// TwinCAT 3 PLC project PLC
// ProgramVersion: 3.1.4026.24
// libraries:
//   Tc2_MC2, * (Beckhoff Automation GmbH)
//   Tc2_Standard, * (Beckhoff Automation GmbH)
//   Tc2_System, * (Beckhoff Automation GmbH)
//   XPlanarApplication, * (Beckhoff Automation LLC)
// project tree:
//   / E_Steps.TcDUT, MAIN.TcPOU, PlcTask.TcTTO
//   Transformation/ ATAN2.TcPOU (not stored), MoverToWorldTransform.TcPOU
// real-time tasks:
//   TASK XPlanar Task_3: cycle T#250us, priority 1, ADS port 350
//   TASK XPlanar Task_4: cycle T#250us, priority 2, ADS port 351
//   TASK XPlanar Task_5: cycle T#250us, priority 3, ADS port 352
//   TASK Job Task: cycle default, priority 4
//   TASK MC-Task (MET): cycle T#2ms, priority 5, ADS port 353
//   TASK MC-Task (MPT): cycle T#10ms, priority 6, ADS port 354
//   TASK PlcTask: cycle T#10ms, priority 20, ADS port 355
// motion (NC):
//   TASK NC-Task 1 SAF: cycle T#2ms, priority 7, ADS port 501
//   TASK NC-Task 1 SVB: cycle T#10ms, priority 12, ADS port 511
//   AXIS CAxis (id 1)
//     Velo: SlowManual=5, FastManual=50
//     OtherSettings: AllowMotionCmdToSlave=true
//     encoder EncType=1
//     drive DrvType=5
//       Analog: TorqueSetpointScale=10, ScaleFactorActTorque=0.1
//       TimeComp: TaskDelayCycles=1
//     controller CtrType=1
//       CtrPara: PriorControlFactor=1
//         Observer: BandWidth=20
// variable links:
//   (this object) <-> NC-Task 1 SAF/Axes/CAxis
//     PlcTask Inputs/MAIN.CAxis.NcToPlc <-> Outputs/ToPlc
//     PlcTask Outputs/MAIN.CAxis.PlcToNc <-> Inputs/FromPlc
//   (this object) <-> XPlanar MC Project/Axes/Mover4330_1
//     PlcTask Inputs/MAIN.Mover._Mover.MCTOPLC/ACT <-> McToPlc/ACT
//     PlcTask Inputs/MAIN.Mover._Mover.MCTOPLC/COORDMODE <-> McToPlc/COORDMODE
//     PlcTask Inputs/MAIN.Mover._Mover.MCTOPLC/SET <-> McToPlc/SET
//     PlcTask Inputs/MAIN.Mover._Mover.MCTOPLC/SETONTRACK <-> McToPlc/SETONTRACK
//     PlcTask Inputs/MAIN.Mover._Mover.MCTOPLC/STD <-> McToPlc/STD
//     PlcTask Outputs/MAIN.Mover._Mover.PLCTOMC/STD <-> PlcToMc/STD
//   (this object) <-> XPlanar MC Project/Groups/Environment
//     PlcTask Inputs/XPlanar.Environment.MCTOPLC_STD <-> McToPlc/STD
//   (this object) <-> XPlanar MC Project/Groups/XPlanar
//     PlcTask Inputs/XPlanar.Group.MCTOPLC_STD <-> McToPlc/STD

CONFIGURATION PLC
    RESOURCE PLC ON TwinCAT3
        TASK PlcTask(INTERVAL := T#10ms, PRIORITY := 20);
        PROGRAM MAIN WITH PlcTask : MAIN;
    END_RESOURCE
END_CONFIGURATION

// ---- E_Steps.TcDUT
{attribute 'qualified_only'}
{attribute 'strict'}
{attribute 'to_string'}
TYPE E_Steps :
(
	init := 0,
    enable,
    enabled,
    moveCenter,
    idle,
    enableExtSp,
    runExtSp,
    error
)UINT;
END_TYPE

// ---- MAIN.TcPOU
PROGRAM MAIN
VAR
   MoverToWorldTransform : MoverToWorldTransform;
   XPlanarTable : FB_Component_XPlanar;
   Mover : FB_XPlanarMover;
   seq : E_Steps;
   subSeq : UDINT;
   
   Position : MoverVector;
   Velocity : MoverVector;
   Acceleration : MoverVector;
   
   CAxisPower : MC_Power;
   CAxis : AXIS_REF;
   a,b : LREAL;
   Exception : __SYSTEM.ExceptionCode;
END_VAR

CASE seq OF
    E_Steps.init:
        ip.Movers[1] := Mover;
        subSeq := 0;
        // wait for manual command to enable
        
    E_Steps.enable:
        IF XplanarTable.EnableMovers().Done THEN
            seq:= E_Steps.enabled;
        END_IF
  
        IF Mover.Error THEN
            seq:= E_Steps.error;
        END_IF
        
   E_Steps.enabled:  
        // wait for manual command to move to center
   E_Steps.moveCenter:
        CASE subSeq OF
            0:
                IF ip.Movers[1].MoveCommand.SquareUp().Done THEN
                     subSeq := 10;
                END_IF
            
            10:
                IF ip.Movers[1].MoveCommand.FreeMove(320, 320, 0).Done THEN
					subSeq := 20;
				END_IF
                
            20:
                IF ip.Movers[1].MoveCommand.VerticalMove(2).Done THEN
					subSeq := 30;
				END_IF
              
            30:   
                IF ip.Movers[1].MoveCommand.TiltA(15).Done THEN
					seq:= E_Steps.idle;
                    subSeq := 0;
				END_IF
        END_CASE
        
        IF Mover.Error THEN
            seq:= E_Steps.error;
        END_IF
        
    E_Steps.idle:
        // wait for manual command to start ext. setpoint gen.
        // Tilt mover in desired direction via motion UI first.
    
    E_Steps.enableExtSp:
        MoverToWorldTransform.MoverX := Mover.ActualPosition.x;
        MoverToWorldTransform.MoverY := Mover.ActualPosition.y;
        MoverToWorldTransform.MoverZ := Mover.ActualPosition.z;
        MoverToWorldTransform.MoverRx := Mover.ActualPosition.a;
        MoverToWorldTransform.MoverRy := -Mover.ActualPosition.b; // invert input of matrix 
        MoverToWorldTransform.MoverRz := Mover.ActualPosition.c;
        seq := E_Steps.runExtSp;
    
    E_Steps.runExtSp:
        MoverToWorldTransform.ToolOffsetRz := CAxis.NcToPlc.ActPos;    
        __TRY
            MoverToWorldTransform();
        __CATCH(Exception) 
            ; 
        __ENDTRY
    
        Position.x := MoverToWorldTransform.WorldX;
        Position.y := MoverToWorldTransform.WorldY;
        Position.z := MoverToWorldTransform.WorldZ;
        Position.a := MoverToWorldTransform.WorldRx;
        Position.b := -MoverToWorldTransform.WorldRy; // find root cause of this inversion to planar tile
        Position.c := MoverToWorldTransform.WorldRz;
        
        Velocity.x := 0;
        Velocity.y := 0;
        Velocity.z := 0;
        Velocity.a := CAxis.NcToPlc.ActVelo; // Needs to be adjusted - calculate velocity in real applications
        Velocity.b := CAxis.NcToPlc.ActVelo; // Needs to be adjusted - calculate velocity in real applications
        Velocity.c := CAxis.NcToPlc.ActVelo;
        
        Acceleration.x := 0;
        Acceleration.y := 0;
        Acceleration.z := 0;
        Acceleration.a := CAxis.NcToPlc.ActAcc;
        Acceleration.b := CAxis.NcToPlc.ActAcc;
        Acceleration.c := CAxis.NcToPlc.ActAcc;
        
        ip.Movers[1].MoveCommand.RunExternalSpAbsoluteMode(Position,Velocity,Acceleration);
END_CASE    


   
CAxisPower(
	Axis:= CAxis, 
	Enable:= TRUE, 
	Enable_Positive:= TRUE, 
	Enable_Negative:= TRUE, 
	Override:= 100.0 );
XplanarTable.CyclicLogic();

a := ATAN2(0,1);
b := ATAN2(1,0);

END_PROGRAM

// ---- Transformation/MoverToWorldTransform.TcPOU
(* ============================================================================
   FUNCTION BLOCK: FB_MoverToWorldTransform
   ----------------------------------------------------------------------------
   PURPOSE:
     Forward transforms a mover tooling position from the mover (local) frame
     into the world coordinate system of the tile.

     Coordinate chain:
       World (Tile) <-- Mover Pose <-- Tool Offset <-- Tool Tip

     Rotation convention: INTRINSIC XYZ (Tait-Bryan)
       Rx applied first (roll around X), then Ry (pitch around Y'),
       then Rz (yaw around Z'').
       Combined matrix: R = Rz * Ry * Rx

     Runs every scan cycle — no enable trigger required.
     All output angles are ABSOLUTE (unbounded, no rollover).

   INPUTS:
     MoverX, MoverY, MoverZ          : Mover position in tile world [mm]
     MoverRx, MoverRy, MoverRz       : Mover orientation in tile world [°]
                                       XYZ intrinsic: Rx first, Rz last
     ToolOffsetX/Y/Z                 : Tool offset in mover-local frame [mm]
     ToolOffsetRx/Ry/Rz             : Tool orientation offset in mover frame [°]
     Reset                           : Clears accumulated angle unwrap history

   OUTPUTS:
     WorldX, WorldY, WorldZ          : Tool tip position in tile world [mm]
     WorldRx, WorldRy, WorldRz       : Tool tip orientation in tile world [°]
                                       ABSOLUTE — never rolls over ±360°
     Error                           : Set TRUE when asin clamp fires (near ±90° pitch)
   ============================================================================ *)

FUNCTION_BLOCK MoverToWorldTransform
VAR_INPUT
    MoverX          : LREAL;
    MoverY          : LREAL;
    MoverZ          : LREAL;
    MoverRx         : LREAL;   (* Roll  around X [°] — applied first  *)
    MoverRy         : LREAL;   (* Pitch around Y [°] — applied second *)
    MoverRz         : LREAL;   (* Yaw   around Z [°] — applied last   *)

    ToolOffsetX     : LREAL;
    ToolOffsetY     : LREAL;
    ToolOffsetZ     : LREAL;
    ToolOffsetRx    : LREAL;
    ToolOffsetRy    : LREAL;
    ToolOffsetRz    : LREAL;

    Reset           : BOOL;
END_VAR

VAR_OUTPUT
    WorldX          : LREAL;
    WorldY          : LREAL;
    WorldZ          : LREAL;
    WorldRx         : LREAL;   (* Absolute, no rollover *)
    WorldRy         : LREAL;   (* Absolute, no rollover *)
    WorldRz         : LREAL;   (* Absolute, no rollover *)
    Error           : BOOL;
END_VAR

VAR
    ResetPrev       : BOOL;

    R_M             : ARRAY[1..3, 1..3] OF LREAL;   (* Mover rotation matrix    *)
    R_T             : ARRAY[1..3, 1..3] OF LREAL;   (* Tool offset rot. matrix  *)
    R_W             : ARRAY[1..3, 1..3] OF LREAL;   (* Combined world rot. matrix *)

    Dx              : LREAL;   (* Tool offset rotated into world frame *)
    Dy              : LREAL;
    Dz              : LREAL;

    RawRx           : LREAL;   (* Wrapped angles extracted from R_W *)
    RawRy           : LREAL;
    RawRz           : LREAL;

    PrevRawRx       : LREAL;
    PrevRawRy       : LREAL;
    PrevRawRz       : LREAL;

    UnwrapOffRx     : LREAL;   (* Accumulated unwrap corrections *)
    UnwrapOffRy     : LREAL;
    UnwrapOffRz     : LREAL;

    FirstCalc       : BOOL := TRUE;

    Cx              : LREAL;   (* Trig intermediates — mover *)
    Sx              : LREAL;
    Cy              : LREAL;
    Sy              : LREAL;
    Cz              : LREAL;
    Sz              : LREAL;

    Cx2             : LREAL;   (* Trig intermediates — tool offset *)
    Sx2             : LREAL;
    Cy2             : LREAL;
    Sy2             : LREAL;
    Cz2             : LREAL;
    Sz2             : LREAL;

    SyWorld         : LREAL;   (* Clamped sin(Ry_world) for gimbal guard *)
END_VAR

VAR CONSTANT
    DEG2RAD         : LREAL := 0.017453292519943295;
    RAD2DEG         : LREAL := 57.29577951308232;
    HALF_TURN       : LREAL := 180.0;
    FULL_TURN       : LREAL := 360.0;
END_VAR

(* ── Reset unwrap history on rising edge ────────────────────────────────────── *)
IF Reset AND NOT ResetPrev THEN
    UnwrapOffRx := 0.0;
    UnwrapOffRy := 0.0;
    UnwrapOffRz := 0.0;
    PrevRawRx   := 0.0;
    PrevRawRy   := 0.0;
    PrevRawRz   := 0.0;
    FirstCalc   := TRUE;
    Error       := FALSE;
END_IF
ResetPrev := Reset;

Error := FALSE;

(* ============================================================================
   MOVER ROTATION MATRIX  R_M = Rz(MoverRz) * Ry(MoverRy) * Rx(MoverRx)
   ============================================================================ *)
Cx := COS(MoverRx * DEG2RAD);
Sx := SIN(MoverRx * DEG2RAD);
Cy := COS(MoverRy * DEG2RAD);
Sy := SIN(MoverRy * DEG2RAD);
Cz := COS(MoverRz * DEG2RAD);
Sz := SIN(MoverRz * DEG2RAD);

R_M[1,1] :=  Cy * Cz;
R_M[1,2] :=  Sx * Sy * Cz - Cx * Sz;
R_M[1,3] :=  Cx * Sy * Cz + Sx * Sz;

R_M[2,1] :=  Cy * Sz;
R_M[2,2] :=  Sx * Sy * Sz + Cx * Cz;
R_M[2,3] :=  Cx * Sy * Sz - Sx * Cz;

R_M[3,1] := -Sy;
R_M[3,2] :=  Sx * Cy;
R_M[3,3] :=  Cx * Cy;

(* ============================================================================
   TOOL OFFSET ROTATION MATRIX  R_T = Rz(ToolOffsetRz) * Ry(ToolOffsetRy) * Rx(ToolOffsetRx)
   ============================================================================ *)
Cx2 := COS(ToolOffsetRx * DEG2RAD);
Sx2 := SIN(ToolOffsetRx * DEG2RAD);
Cy2 := COS(ToolOffsetRy * DEG2RAD);
Sy2 := SIN(ToolOffsetRy * DEG2RAD);
Cz2 := COS(ToolOffsetRz * DEG2RAD);
Sz2 := SIN(ToolOffsetRz * DEG2RAD);

R_T[1,1] :=  Cy2 * Cz2;
R_T[1,2] :=  Sx2 * Sy2 * Cz2 - Cx2 * Sz2;
R_T[1,3] :=  Cx2 * Sy2 * Cz2 + Sx2 * Sz2;

R_T[2,1] :=  Cy2 * Sz2;
R_T[2,2] :=  Sx2 * Sy2 * Sz2 + Cx2 * Cz2;
R_T[2,3] :=  Cx2 * Sy2 * Sz2 - Sx2 * Cz2;

R_T[3,1] := -Sy2;
R_T[3,2] :=  Sx2 * Cy2;
R_T[3,3] :=  Cx2 * Cy2;

(* ============================================================================
   COMBINED WORLD ROTATION  R_W = R_M * R_T
   ============================================================================ *)
R_W[1,1] := R_M[1,1]*R_T[1,1] + R_M[1,2]*R_T[2,1] + R_M[1,3]*R_T[3,1];
R_W[1,2] := R_M[1,1]*R_T[1,2] + R_M[1,2]*R_T[2,2] + R_M[1,3]*R_T[3,2];
R_W[1,3] := R_M[1,1]*R_T[1,3] + R_M[1,2]*R_T[2,3] + R_M[1,3]*R_T[3,3];

R_W[2,1] := R_M[2,1]*R_T[1,1] + R_M[2,2]*R_T[2,1] + R_M[2,3]*R_T[3,1];
R_W[2,2] := R_M[2,1]*R_T[1,2] + R_M[2,2]*R_T[2,2] + R_M[2,3]*R_T[3,2];
R_W[2,3] := R_M[2,1]*R_T[1,3] + R_M[2,2]*R_T[2,3] + R_M[2,3]*R_T[3,3];

R_W[3,1] := R_M[3,1]*R_T[1,1] + R_M[3,2]*R_T[2,1] + R_M[3,3]*R_T[3,1];
R_W[3,2] := R_M[3,1]*R_T[1,2] + R_M[3,2]*R_T[2,2] + R_M[3,3]*R_T[3,2];
R_W[3,3] := R_M[3,1]*R_T[1,3] + R_M[3,2]*R_T[2,3] + R_M[3,3]*R_T[3,3];

(* ============================================================================
   WORLD POSITION
   Tool offset translated by R_M into the world frame, added to mover position
   ============================================================================ *)
Dx := R_M[1,1]*ToolOffsetX + R_M[1,2]*ToolOffsetY + R_M[1,3]*ToolOffsetZ;
Dy := R_M[2,1]*ToolOffsetX + R_M[2,2]*ToolOffsetY + R_M[2,3]*ToolOffsetZ;
Dz := R_M[3,1]*ToolOffsetX + R_M[3,2]*ToolOffsetY + R_M[3,3]*ToolOffsetZ;

WorldX := MoverX + Dx;
WorldY := MoverY + Dy;
WorldZ := MoverZ + Dz;

(* ============================================================================
   EXTRACT XYZ EULER ANGLES FROM R_W
     Ry = asin( -R_W[3,1] )
     Rx = atan2(  R_W[3,2],  R_W[3,3] )
     Rz = atan2(  R_W[2,1],  R_W[1,1] )
   R_W[3,1] clamped to [-1, 1] to prevent NaN at the ±90° pitch singularity
   ============================================================================ *)
SyWorld := R_W[3,1];
IF SyWorld >  1.0 THEN SyWorld :=  1.0; Error := TRUE; END_IF
IF SyWorld < -1.0 THEN SyWorld := -1.0; Error := TRUE; END_IF

RawRy := ASIN(-SyWorld)            * RAD2DEG;
RawRx := ATAN2(R_W[3,2], R_W[3,3]) * RAD2DEG;
RawRz := ATAN2(R_W[2,1], R_W[1,1]) * RAD2DEG;

(* ============================================================================
   ANGLE UNWRAP — prevent ±360° rollover
   ASIN output is bounded to [-90, +90] and ATAN2 to [-180, +180], so a raw
   angle can jump at most 360° per cycle. A single IF per axis is sufficient.
   ============================================================================ *)
IF FirstCalc THEN
    PrevRawRx   := RawRx;
    PrevRawRy   := RawRy;
    PrevRawRz   := RawRz;
    UnwrapOffRx := 0.0;
    UnwrapOffRy := 0.0;
    UnwrapOffRz := 0.0;
    FirstCalc   := FALSE;
ELSE
    IF (RawRx - PrevRawRx) >  HALF_TURN THEN UnwrapOffRx := UnwrapOffRx - FULL_TURN; END_IF
    IF (RawRx - PrevRawRx) < -HALF_TURN THEN UnwrapOffRx := UnwrapOffRx + FULL_TURN; END_IF

    IF (RawRy - PrevRawRy) >  HALF_TURN THEN UnwrapOffRy := UnwrapOffRy - FULL_TURN; END_IF
    IF (RawRy - PrevRawRy) < -HALF_TURN THEN UnwrapOffRy := UnwrapOffRy + FULL_TURN; END_IF

    IF (RawRz - PrevRawRz) >  HALF_TURN THEN UnwrapOffRz := UnwrapOffRz - FULL_TURN; END_IF
    IF (RawRz - PrevRawRz) < -HALF_TURN THEN UnwrapOffRz := UnwrapOffRz + FULL_TURN; END_IF

    PrevRawRx := RawRx;
    PrevRawRy := RawRy;
    PrevRawRz := RawRz;
END_IF

(* ── Absolute output angles ─────────────────────────────────────────────────── *)
WorldRx := RawRx + UnwrapOffRx;
WorldRy := RawRy + UnwrapOffRy;
WorldRz := RawRz + UnwrapOffRz;

END_FUNCTION_BLOCK
